{attribute 'qualified_only'}
{attribute 'strict'}
TYPE E_ControlMode :
(
	Position 	:= 0,
	Speed	 	:= 1
)
BYTE;
END_TYPE

(* stored: Version 1.1.0.1, ProductVersion 3.1.4024.12
   DUT E_ControlMode: Id {b0885657-7658-0924-181e-609954663d8a} *)
